// Block: HW_Const_Values

DATA_BLOCK HW_Const_Values
VERSION : 0.1
   NON_RETAIN
   VAR
      CU2_PN_IODevice : HW_DEVICE;
      CU2_PN : HW_INTERFACE;
      CU2_PN_Port_1 : HW_INTERFACE;
      CU2_PN_Port_2 : HW_INTERFACE;
      CU2_PN_585A1_ModuleAccessPoint : HW_SUBMODULE;
      CU2_PN_1190A1_ModuleAccessPoint : HW_SUBMODULE;
      CU2_PN_1300A1_ModuleAccessPoint : HW_SUBMODULE;
      CU2_PN_830A1_ModuleAccessPoint : HW_SUBMODULE;
      CU2_PN_1 : HW_INTERFACE;
      CU2_PN_Port_1_1 : HW_INTERFACE;
      CU2_PN_Port_2_1 : HW_INTERFACE;
      CU2_PN_2 : HW_INTERFACE;
      CU2_PN_Port_1_2 : HW_INTERFACE;
      CU2_PN_Port_2_2 : HW_INTERFACE;
      CU2_PN_3 : HW_INTERFACE;
      CU2_PN_Port_1_3 : HW_INTERFACE;
      CU2_PN_Port_2_3 : HW_INTERFACE;
      Local_PROFINET_interface_GBIT_3 : HW_INTERFACE;
      Local_PROFINET_interface_GBIT_3_Port_1 : HW_INTERFACE;
      Local_412A1 : HW_SUBMODULE;
      Local_413A1 : HW_SUBMODULE;
      Local_413A2 : HW_SUBMODULE;
      Local_414A1 : HW_SUBMODULE;
      Local_415A1 : HW_SUBMODULE;
      Local_415A2 : HW_SUBMODULE;
      HW_460A1_JB001_Proxy : HW_SUBMODULE;
      HW_460A1_JB001_IODevice : HW_DEVICE;
      HW_460A1_JB001_Head : HW_SUBMODULE;
      HW_460A1_JB001_460A1_X1 : HW_INTERFACE;
      HW_460A1_JB001_479A3 : HW_SUBMODULE;
      HW_460A1_JB001_479A4 : HW_SUBMODULE;
      HW_460A1_JB001_480A1 : HW_SUBMODULE;
      HW_460A1_JB001_480A2 : HW_SUBMODULE;
      HW_460A1_JB001_482A1 : HW_SUBMODULE;
      HW_460A1_JB001_482A2 : HW_SUBMODULE;
      HW_460A1_JB001_Server_module_1 : HW_SUBMODULE;
      HW_460A1_JB001_464A1 : HW_SUBMODULE;
      HW_460A1_JB001_470A2 : HW_SUBMODULE;
      HW_460A1_JB001_470A1 : HW_SUBMODULE;
      HW_460A1_JB001_463A1 : HW_SUBMODULE;
      HW_460A1_JB001_460A1_X1_Port_2 : HW_INTERFACE;
      HW_460A1_JB001_460A1_X1_Port_1 : HW_INTERFACE;
      HW_460A1_JB001_465A1 : HW_SUBMODULE;
      HW_460A1_JB001_468A1 : HW_SUBMODULE;
      HW_460A1_JB001_468A2 : HW_SUBMODULE;
      HW_460A1_JB001_468A3 : HW_SUBMODULE;
      HW_460A1_JB001_468A4 : HW_SUBMODULE;
      HW_460A1_JB001_468A5 : HW_SUBMODULE;
      HW_460A1_JB001_468A6 : HW_SUBMODULE;
      HW_460A1_JB001_468A7 : HW_SUBMODULE;
      HW_460A1_JB001_468A8 : HW_SUBMODULE;
      HW_460A1_JB001_471A1 : HW_SUBMODULE;
      HW_460A1_JB001_471A2 : HW_SUBMODULE;
      HW_460A1_JB001_472A1 : HW_SUBMODULE;
      HW_460A1_JB001_474A1 : HW_SUBMODULE;
      HW_460A1_JB001_474A2 : HW_SUBMODULE;
      HW_460A1_JB001_474A3 : HW_SUBMODULE;
      HW_460A1_JB001_474A4 : HW_SUBMODULE;
      HW_460A1_JB001_474A5 : HW_SUBMODULE;
      HW_460A1_JB001_474A6 : HW_SUBMODULE;
      HW_460A1_JB001_474A7 : HW_SUBMODULE;
      HW_460A1_JB001_474A8 : HW_SUBMODULE;
      HW_460A1_JB001_475A1 : HW_SUBMODULE;
      HW_460A1_JB001_475A2 : HW_SUBMODULE;
      HW_460A1_JB001_475A3 : HW_SUBMODULE;
      HW_460A1_JB001_475A4 : HW_SUBMODULE;
      HW_460A1_JB001_475A5 : HW_SUBMODULE;
      HW_460A1_JB001_475A6 : HW_SUBMODULE;
      HW_460A1_JB001_475A7 : HW_SUBMODULE;
      HW_460A1_JB001_475A8 : HW_SUBMODULE;
      HW_460A1_JB001_476A1 : HW_SUBMODULE;
      HW_460A1_JB001_476A2 : HW_SUBMODULE;
      HW_460A1_JB001_476A3 : HW_SUBMODULE;
      HW_460A1_JB001_476A4 : HW_SUBMODULE;
      HW_460A1_JB001_476A5 : HW_SUBMODULE;
      HW_460A1_JB001_476A6 : HW_SUBMODULE;
      HW_460A1_JB001_478A1 : HW_SUBMODULE;
      HW_460A1_JB001_478A2 : HW_SUBMODULE;
      HW_460A1_JB001_478A3 : HW_SUBMODULE;
      HW_460A1_JB001_478A4 : HW_SUBMODULE;
      HW_460A1_JB001_478A5 : HW_SUBMODULE;
      HW_460A1_JB001_478A6 : HW_SUBMODULE;
      HW_460A1_JB001_478A7 : HW_SUBMODULE;
      HW_460A1_JB001_478A8 : HW_SUBMODULE;
      HW_460A1_JB001_479A1 : HW_SUBMODULE;
      HW_460A1_JB001_479A2 : HW_SUBMODULE;
      HW_490A1_JB301_Proxy : HW_SUBMODULE;
      HW_490A1_JB301_IODevice : HW_DEVICE;
      HW_490A1_JB301_Head : HW_SUBMODULE;
      HW_490A1_JB301_PROFINET_interface : HW_INTERFACE;
      HW_490A1_JB301_495A2 : HW_SUBMODULE;
      HW_490A1_JB301_495A1 : HW_SUBMODULE;
      HW_490A1_JB301_PROFINET_interface_Port_2 : HW_INTERFACE;
      HW_490A1_JB301_PROFINET_interface_Port_1 : HW_INTERFACE;
      HW_510A1_JB302_Proxy : HW_SUBMODULE;
      HW_510A1_JB302_IODevice : HW_DEVICE;
      HW_510A1_JB302_Head : HW_SUBMODULE;
      HW_510A1_JB302_PROFINET_interface : HW_INTERFACE;
      HW_510A1_JB302_515A2 : HW_SUBMODULE;
      HW_510A1_JB302_515A1 : HW_SUBMODULE;
      HW_510A1_JB302_513A1 : HW_SUBMODULE;
      HW_510A1_JB302_512A1 : HW_SUBMODULE;
      HW_510A1_JB302_PROFINET_interface_Port_2 : HW_INTERFACE;
      HW_510A1_JB302_PROFINET_interface_Port_1 : HW_INTERFACE;
      HW_530A1_JB305_Proxy : HW_SUBMODULE;
      HW_530A1_JB305_IODevice : HW_DEVICE;
      HW_530A1_JB305_Head : HW_SUBMODULE;
      HW_530A1_JB305_PROFINET_interface : HW_INTERFACE;
      HW_530A1_JB305_542A3 : HW_SUBMODULE;
      HW_530A1_JB305_542A2 : HW_SUBMODULE;
      HW_530A1_JB305_542A1 : HW_SUBMODULE;
      HW_530A1_JB305_540A2 : HW_SUBMODULE;
      HW_530A1_JB305_540A1 : HW_SUBMODULE;
      HW_530A1_JB305_538A6 : HW_SUBMODULE;
      HW_530A1_JB305_538A5 : HW_SUBMODULE;
      HW_530A1_JB305_538A4 : HW_SUBMODULE;
      HW_530A1_JB305_538A3 : HW_SUBMODULE;
      HW_530A1_JB305_538A2 : HW_SUBMODULE;
      HW_530A1_JB305_538A1 : HW_SUBMODULE;
      HW_530A1_JB305_537A1 : HW_SUBMODULE;
      HW_530A1_JB305_536A1 : HW_SUBMODULE;
      HW_530A1_JB305_535A2 : HW_SUBMODULE;
      HW_530A1_JB305_535A1 : HW_SUBMODULE;
      HW_530A1_JB305_533A1 : HW_SUBMODULE;
      HW_530A1_JB305_PROFINET_interface_Port_2 : HW_INTERFACE;
      HW_530A1_JB305_PROFINET_interface_Port_1 : HW_INTERFACE;
      HW_550A1_JB306_Proxy : HW_SUBMODULE;
      HW_550A1_JB306_IODevice : HW_DEVICE;
      HW_550A1_JB306_Head : HW_SUBMODULE;
      HW_550A1_JB306_PROFINET_interface : HW_INTERFACE;
      HW_550A1_JB306_562A3 : HW_SUBMODULE;
      HW_550A1_JB306_562A2 : HW_SUBMODULE;
      HW_550A1_JB306_562A1 : HW_SUBMODULE;
      HW_550A1_JB306_560A2 : HW_SUBMODULE;
      HW_550A1_JB306_560A1 : HW_SUBMODULE;
      HW_550A1_JB306_558A6 : HW_SUBMODULE;
      HW_550A1_JB306_558A5 : HW_SUBMODULE;
      HW_550A1_JB306_558A4 : HW_SUBMODULE;
      HW_550A1_JB306_558A3 : HW_SUBMODULE;
      HW_550A1_JB306_558A2 : HW_SUBMODULE;
      HW_550A1_JB306_558A1 : HW_SUBMODULE;
      HW_550A1_JB306_556A1 : HW_SUBMODULE;
      HW_550A1_JB306_555A1 : HW_SUBMODULE;
      HW_550A1_JB306_552A1 : HW_SUBMODULE;
      HW_550A1_JB306_PROFINET_interface_Port_2 : HW_INTERFACE;
      HW_550A1_JB306_PROFINET_interface_Port_1 : HW_INTERFACE;
      CU1_PN_IODevice : HW_DEVICE;
      CU1_PN : HW_INTERFACE;
      CU1_PN_Port_1 : HW_INTERFACE;
      CU1_PN_Port_2 : HW_INTERFACE;
      CU1_PN_580A1_ModuleAccessPoint : HW_SUBMODULE;
      CU1_PN_740A1_1_ModuleAccessPoint : HW_SUBMODULE;
      CU1_PN_740A1_2_ModuleAccessPoint : HW_SUBMODULE;
      CU1_PN_690A1_1_ModuleAccessPoint : HW_SUBMODULE;
      CU1_PN_690A1_2_ModuleAccessPoint : HW_SUBMODULE;
      CU1_PN_890A1_1_ModuleAccessPoint : HW_SUBMODULE;
      CU1_PN_890A1_2_ModuleAccessPoint : HW_SUBMODULE;
      CU1_PN_1 : HW_INTERFACE;
      CU1_PN_Port_1_1 : HW_INTERFACE;
      CU1_PN_Port_2_1 : HW_INTERFACE;
      CU1_PN_2 : HW_INTERFACE;
      CU1_PN_Port_1_2 : HW_INTERFACE;
      CU1_PN_Port_2_2 : HW_INTERFACE;
      CU1_PN_3 : HW_INTERFACE;
      CU1_PN_Port_1_3 : HW_INTERFACE;
      CU1_PN_Port_2_3 : HW_INTERFACE;
      CU3_PROFINET_interface_IODevice : HW_DEVICE;
      CU3_PROFINET_interface : HW_INTERFACE;
      CU3_PROFINET_interface_Port_1 : HW_INTERFACE;
      CU3_PROFINET_interface_Port_2 : HW_INTERFACE;
      CU3_PROFINET_interface_590A1_ModuleAccessPoint : HW_SUBMODULE;
      CU3_PROFINET_interface_590A1_SIEMENS_telegram_393 : HW_SUBMODULE;
      CU3_PROFINET_interface_1410A1_1_ModuleAccessPoint : HW_SUBMODULE;
      CU3_PROFINET_interface_1410A1_1_PROFIsafe_telegram_30 : HW_SUBMODULE;
      CU3_PROFINET_interface_1410A1_2_ModuleAccessPoint : HW_SUBMODULE;
      CU3_PROFINET_interface_1410A1_2_PROFIsafe_telegram_30 : HW_SUBMODULE;
      CU3_PROFINET_interface_1430A1_1_ModuleAccessPoint : HW_SUBMODULE;
      CU3_PROFINET_interface_1430A1_1_PROFIsafe_telegram_30 : HW_SUBMODULE;
      CU3_PROFINET_interface_1430A1_2_ModuleAccessPoint : HW_SUBMODULE;
      CU3_PROFINET_interface_1430A1_2_PROFIsafe_telegram_30 : HW_SUBMODULE;
      CU3_PROFINET_interface_1260A1_1_ModuleAccessPoint : HW_SUBMODULE;
      CU3_PROFINET_interface_1260A1_1_PROFIsafe_telegram_30 : HW_SUBMODULE;
      CU3_PROFINET_interface_1260A1_2_ModuleAccessPoint : HW_SUBMODULE;
      CU3_PROFINET_interface_1260A1_2_PROFIsafe_telegram_30 : HW_SUBMODULE;
      CU3_PROFINET_interface_1 : HW_INTERFACE;
      CU3_PROFINET_interface_Port_1_1 : HW_INTERFACE;
      CU3_PROFINET_interface_Port_2_1 : HW_INTERFACE;
      CU3_PROFINET_interface_2 : HW_INTERFACE;
      CU3_PROFINET_interface_Port_1_2 : HW_INTERFACE;
      CU3_PROFINET_interface_Port_2_2 : HW_INTERFACE;
      CU3_PROFINET_interface_3 : HW_INTERFACE;
      CU3_PROFINET_interface_Port_1_3 : HW_INTERFACE;
      CU3_PROFINET_interface_Port_2_3 : HW_INTERFACE;
      CU4_PN_IODevice : HW_DEVICE;
      CU4_PN : HW_INTERFACE;
      CU4_PN_Port_1 : HW_INTERFACE;
      CU4_PN_Port_2 : HW_INTERFACE;
      CU4_PN_595A1_ModuleAccessPoint : HW_SUBMODULE;
      CU4_PN_595A1_SIEMENS_telegram_393 : HW_SUBMODULE;
      CU4_PN_980A1_1_ModuleAccessPoint : HW_SUBMODULE;
      CU4_PN_980A1_1_PROFIsafe_telegram_30 : HW_SUBMODULE;
      CU4_PN_980A1_2_ModuleAccessPoint : HW_SUBMODULE;
      CU4_PN_980A1_2_PROFIsafe_telegram_30 : HW_SUBMODULE;
      CU4_PN_1030A1_1_ModuleAccessPoint : HW_SUBMODULE;
      CU4_PN_1030A1_1_PROFIsafe_telegram_30 : HW_SUBMODULE;
      CU4_PN_1030A1_2_ModuleAccessPoint : HW_SUBMODULE;
      CU4_PN_1030A1_2_PROFIsafe_telegram_30 : HW_SUBMODULE;
      CU4_PN_1070A1_1_ModuleAccessPoint : HW_SUBMODULE;
      CU4_PN_1070A1_1_PROFIsafe_telegram_30 : HW_SUBMODULE;
      CU4_PN_1070A1_2_ModuleAccessPoint : HW_SUBMODULE;
      CU4_PN_1070A1_2_PROFIsafe_telegram_30 : HW_SUBMODULE;
      CU4_PN_1 : HW_INTERFACE;
      CU4_PN_Port_1_1 : HW_INTERFACE;
      CU4_PN_Port_2_1 : HW_INTERFACE;
      CU4_PN_2 : HW_INTERFACE;
      CU4_PN_Port_1_2 : HW_INTERFACE;
      CU4_PN_Port_2_2 : HW_INTERFACE;
      CU4_PN_3 : HW_INTERFACE;
      CU4_PN_Port_1_3 : HW_INTERFACE;
      CU4_PN_Port_2_3 : HW_INTERFACE;
      CU5_PN_IODevice : HW_DEVICE;
      CU5_PN : HW_INTERFACE;
      CU5_PN_Port_1 : HW_INTERFACE;
      CU5_PN_Port_2 : HW_INTERFACE;
      CU5_PN_600A1_ModuleAccessPoint : HW_SUBMODULE;
      CU5_PN_600A1_SIEMENS_telegram_393 : HW_SUBMODULE;
      CU5_PN_1950A1_ModuleAccessPoint : HW_SUBMODULE;
      CU5_PN_1950A1_SIEMENS_telegram_111 : HW_SUBMODULE;
      CU5_PN_1950A1_PROFIsafe_telegram_30 : HW_SUBMODULE;
      CU5_PN_1480A1_1_ModuleAccessPoint : HW_SUBMODULE;
      CU5_PN_1480A1_1_PROFIsafe_telegram_30 : HW_SUBMODULE;
      CU5_PN_1480A1_2_ModuleAccessPoint : HW_SUBMODULE;
      CU5_PN_1480A1_2_PROFIsafe_telegram_30 : HW_SUBMODULE;
      CU5_PN_1560A1_1_ModuleAccessPoint : HW_SUBMODULE;
      CU5_PN_1560A1_1_SIEMENS_telegram_111 : HW_SUBMODULE;
      CU5_PN_1560A1_1_PROFIsafe_telegram_30 : HW_SUBMODULE;
      CU5_PN_1560A1_2_ModuleAccessPoint : HW_SUBMODULE;
      CU5_PN_1560A1_2_SIEMENS_telegram_111 : HW_SUBMODULE;
      CU5_PN_1560A1_2_PROFIsafe_telegram_30 : HW_SUBMODULE;
      CU5_PN_1 : HW_INTERFACE;
      CU5_PN_Port_1_1 : HW_INTERFACE;
      CU5_PN_Port_2_1 : HW_INTERFACE;
      CU5_PN_2 : HW_INTERFACE;
      CU5_PN_Port_1_2 : HW_INTERFACE;
      CU5_PN_Port_2_2 : HW_INTERFACE;
      CU5_PN_3 : HW_INTERFACE;
      CU5_PN_Port_1_3 : HW_INTERFACE;
      CU5_PN_Port_2_3 : HW_INTERFACE;
      CU6_PN_IODevice : HW_DEVICE;
      CU6_PN : HW_INTERFACE;
      CU6_PN_Port_1 : HW_INTERFACE;
      CU6_PN_Port_2 : HW_INTERFACE;
      CU6_PN_605A1_ModuleAccessPoint : HW_SUBMODULE;
      CU6_PN_605A1_SIEMENS_telegram_393 : HW_SUBMODULE;
      CU6_PN_1990A1_1_ModuleAccessPoint : HW_SUBMODULE;
      CU6_PN_1990A1_1_PROFIsafe_telegram_30 : HW_SUBMODULE;
      CU6_PN_1990A1_2_ModuleAccessPoint : HW_SUBMODULE;
      CU6_PN_1990A1_2_PROFIsafe_telegram_30 : HW_SUBMODULE;
      CU6_PN_2100A1_1_ModuleAccessPoint : HW_SUBMODULE;
      CU6_PN_2100A1_1_SIEMENS_telegram_1 : HW_SUBMODULE;
      CU6_PN_2100A1_1_PROFIsafe_telegram_30 : HW_SUBMODULE;
      CU6_PN_2100A1_2_ModuleAccessPoint : HW_SUBMODULE;
      CU6_PN_2100A1_2_SIEMENS_telegram_1 : HW_SUBMODULE;
      CU6_PN_2100A1_2_PROFIsafe_telegram_30 : HW_SUBMODULE;
      CU6_PN_1840A1_1_ModuleAccessPoint : HW_SUBMODULE;
      CU6_PN_1840A1_1_PROFIsafe_telegram_30 : HW_SUBMODULE;
      CU6_PN_1840A1_2_ModuleAccessPoint : HW_SUBMODULE;
      CU6_PN_1840A1_2_PROFIsafe_telegram_30 : HW_SUBMODULE;
      CU6_PN_1 : HW_INTERFACE;
      CU6_PN_Port_1_1 : HW_INTERFACE;
      CU6_PN_Port_2_1 : HW_INTERFACE;
      CU6_PN_2 : HW_INTERFACE;
      CU6_PN_Port_1_2 : HW_INTERFACE;
      CU6_PN_Port_2_2 : HW_INTERFACE;
      CU6_PN_3 : HW_INTERFACE;
      CU6_PN_Port_1_3 : HW_INTERFACE;
      CU6_PN_Port_2_3 : HW_INTERFACE;
      CU7_PN_IODevice : HW_DEVICE;
      CU7_PN : HW_INTERFACE;
      CU7_PN_Port_1 : HW_INTERFACE;
      CU7_PN_Port_2 : HW_INTERFACE;
      CU7_PN_610A1_ModuleAccessPoint : HW_SUBMODULE;
      CU7_PN_610A1_SIEMENS_telegram_393 : HW_SUBMODULE;
      CU7_PN_2310A1_1_ModuleAccessPoint : HW_SUBMODULE;
      CU7_PN_2310A1_1_SIEMENS_telegram_111 : HW_SUBMODULE;
      CU7_PN_2310A1_1_PROFIsafe_telegram_30 : HW_SUBMODULE;
      CU7_PN_2310A1_2_ModuleAccessPoint : HW_SUBMODULE;
      CU7_PN_2310A1_2_SIEMENS_telegram_111 : HW_SUBMODULE;
      CU7_PN_2310A1_2_PROFIsafe_telegram_30 : HW_SUBMODULE;
      CU7_PN_2260A1_1_ModuleAccessPoint : HW_SUBMODULE;
      CU7_PN_2260A1_1_PROFIsafe_telegram_30 : HW_SUBMODULE;
      CU7_PN_2260A1_2_ModuleAccessPoint : HW_SUBMODULE;
      CU7_PN_2260A1_2_PROFIsafe_telegram_30 : HW_SUBMODULE;
      CU7_PN_2140A1_1_ModuleAccessPoint : HW_SUBMODULE;
      CU7_PN_2140A1_1_SIEMENS_telegram_111 : HW_SUBMODULE;
      CU7_PN_2140A1_1_PROFIsafe_telegram_30 : HW_SUBMODULE;
      CU7_PN_2140A1_2_ModuleAccessPoint : HW_SUBMODULE;
      CU7_PN_2140A1_2_SIEMENS_telegram_111 : HW_SUBMODULE;
      CU7_PN_2140A1_2_PROFIsafe_telegram_30 : HW_SUBMODULE;
      CU7_PN_1 : HW_INTERFACE;
      CU7_PN_Port_1_1 : HW_INTERFACE;
      CU7_PN_Port_2_1 : HW_INTERFACE;
      CU7_PN_2 : HW_INTERFACE;
      CU7_PN_Port_1_2 : HW_INTERFACE;
      CU7_PN_Port_2_2 : HW_INTERFACE;
      CU7_PN_3 : HW_INTERFACE;
      CU7_PN_Port_1_3 : HW_INTERFACE;
      CU7_PN_Port_2_3 : HW_INTERFACE;
      CU8_PN_IODevice : HW_DEVICE;
      CU8_PN : HW_INTERFACE;
      CU8_PN_Port_1 : HW_INTERFACE;
      CU8_PN_Port_2 : HW_INTERFACE;
      CU8_PN_615A1_ModuleAccessPoint : HW_SUBMODULE;
      CU8_PN_615A1_SIEMENS_telegram_393 : HW_SUBMODULE;
      CU8_PN_2390A1_1_ModuleAccessPoint : HW_SUBMODULE;
      CU8_PN_2390A1_1_PROFIsafe_telegram_30 : HW_SUBMODULE;
      CU8_PN_2390A1_2_ModuleAccessPoint : HW_SUBMODULE;
      CU8_PN_2390A1_2_PROFIsafe_telegram_30 : HW_SUBMODULE;
      CU8_PN_2430A1_1_ModuleAccessPoint : HW_SUBMODULE;
      CU8_PN_2430A1_1_PROFIsafe_telegram_30 : HW_SUBMODULE;
      CU8_PN_2430A1_2_ModuleAccessPoint : HW_SUBMODULE;
      CU8_PN_2430A1_2_PROFIsafe_telegram_30 : HW_SUBMODULE;
      CU8_PN_2350A1_1_ModuleAccessPoint : HW_SUBMODULE;
      CU8_PN_2350A1_1_PROFIsafe_telegram_30 : HW_SUBMODULE;
      CU8_PN_2350A1_2_ModuleAccessPoint : HW_SUBMODULE;
      CU8_PN_2350A1_2_PROFIsafe_telegram_30 : HW_SUBMODULE;
      CU8_PN_640A1_ModuleAccessPoint : HW_SUBMODULE;
      CU8_PN_640A1_SIEMENS_telegram_370 : HW_SUBMODULE;
      CU8_PN_1 : HW_INTERFACE;
      CU8_PN_Port_1_1 : HW_INTERFACE;
      CU8_PN_Port_2_1 : HW_INTERFACE;
      CU8_PN_2 : HW_INTERFACE;
      CU8_PN_Port_1_2 : HW_INTERFACE;
      CU8_PN_Port_2_2 : HW_INTERFACE;
      CU8_PN_3 : HW_INTERFACE;
      CU8_PN_Port_1_3 : HW_INTERFACE;
      CU8_PN_Port_2_3 : HW_INTERFACE;
      HW_1008P1_Proxy : HW_SUBMODULE;
      HW_1008P1_IODevice : HW_DEVICE;
      HW_1008P1_Interface : HW_INTERFACE;
      HW_1008P1_Interface_Port_1 : HW_INTERFACE;
      HW_1008P1_Interface_Port_2 : HW_INTERFACE;
      HW_1008P1_Head : HW_SUBMODULE;
      HW_1008P1_EO_Multiturn_1 : HW_SUBMODULE;
      HW_1008P1_Telegram_81_DI_DO : HW_SUBMODULE;
      HW_1008P1_EO_Multiturn_1_Parameter_Access_Point : HW_SUBMODULE;
      HW_1004P1_Proxy : HW_SUBMODULE;
      HW_1004P1_IODevice : HW_DEVICE;
      HW_1004P1_Interface : HW_INTERFACE;
      HW_1004P1_Interface_Port_1 : HW_INTERFACE;
      HW_1004P1_Interface_Port_2 : HW_INTERFACE;
      HW_1004P1_Head : HW_SUBMODULE;
      HW_1004P1_EO_Multiturn_1 : HW_SUBMODULE;
      HW_1004P1_Telegram_81_DI_DO : HW_SUBMODULE;
      HW_1004P1_EO_Multiturn_1_Parameter_Access_Point : HW_SUBMODULE;
      HW_994P1_Proxy : HW_SUBMODULE;
      HW_994P1_IODevice : HW_DEVICE;
      HW_994P1_Interface : HW_INTERFACE;
      HW_994P1_Interface_Port_1 : HW_INTERFACE;
      HW_994P1_Interface_Port_2 : HW_INTERFACE;
      HW_994P1_Head : HW_SUBMODULE;
      HW_994P1_EO_Multiturn_1 : HW_SUBMODULE;
      HW_994P1_Telegram_81_DI_DO : HW_SUBMODULE;
      HW_994P1_EO_Multiturn_1_Parameter_Access_Point : HW_SUBMODULE;
      HW_984P1_Proxy : HW_SUBMODULE;
      HW_984P1_IODevice : HW_DEVICE;
      HW_984P1_Interface : HW_INTERFACE;
      HW_984P1_Interface_Port_1 : HW_INTERFACE;
      HW_984P1_Interface_Port_2 : HW_INTERFACE;
      HW_984P1_Head : HW_SUBMODULE;
      HW_984P1_EO_Multiturn_1 : HW_SUBMODULE;
      HW_984P1_Telegram_81_DI_DO : HW_SUBMODULE;
      HW_984P1_EO_Multiturn_1_Parameter_Access_Point : HW_SUBMODULE;
      HW_1868P1_Proxy : HW_SUBMODULE;
      HW_1868P1_IODevice : HW_DEVICE;
      HW_1868P1_Interface : HW_INTERFACE;
      HW_1868P1_Interface_Port_1 : HW_INTERFACE;
      HW_1868P1_Interface_Port_2 : HW_INTERFACE;
      HW_1868P1_Head : HW_SUBMODULE;
      HW_1868P1_EO_Multiturn_1 : HW_SUBMODULE;
      HW_1868P1_Telegram_81_DI_DO : HW_SUBMODULE;
      HW_1868P1_EO_Multiturn_1_Parameter_Access_Point : HW_SUBMODULE;
      HW_1863P1_Proxy : HW_SUBMODULE;
      HW_1863P1_IODevice : HW_DEVICE;
      HW_1863P1_Interface : HW_INTERFACE;
      HW_1863P1_Interface_Port_1 : HW_INTERFACE;
      HW_1863P1_Interface_Port_2 : HW_INTERFACE;
      HW_1863P1_Head : HW_SUBMODULE;
      HW_1863P1_EO_Multiturn_1 : HW_SUBMODULE;
      HW_1863P1_Telegram_81_DI_DO : HW_SUBMODULE;
      HW_1863P1_EO_Multiturn_1_Parameter_Access_Point : HW_SUBMODULE;
      HW_1858P1_Proxy : HW_SUBMODULE;
      HW_1858P1_IODevice : HW_DEVICE;
      HW_1858P1_Interface : HW_INTERFACE;
      HW_1858P1_Interface_Port_1 : HW_INTERFACE;
      HW_1858P1_Interface_Port_2 : HW_INTERFACE;
      HW_1858P1_Head : HW_SUBMODULE;
      HW_1858P1_EO_Multiturn_1 : HW_SUBMODULE;
      HW_1858P1_Telegram_81_DI_DO : HW_SUBMODULE;
      HW_1858P1_EO_Multiturn_1_Parameter_Access_Point : HW_SUBMODULE;
      HW_1853P1_Proxy : HW_SUBMODULE;
      HW_1853P1_IODevice : HW_DEVICE;
      HW_1853P1_Interface : HW_INTERFACE;
      HW_1853P1_Interface_Port_1 : HW_INTERFACE;
      HW_1853P1_Interface_Port_2 : HW_INTERFACE;
      HW_1853P1_Head : HW_SUBMODULE;
      HW_1853P1_EO_Multiturn_1 : HW_SUBMODULE;
      HW_1853P1_Telegram_81_DI_DO : HW_SUBMODULE;
      HW_1853P1_EO_Multiturn_1_Parameter_Access_Point : HW_SUBMODULE;
      HW_1844P1_Proxy : HW_SUBMODULE;
      HW_1844P1_IODevice : HW_DEVICE;
      HW_1844P1_Interface : HW_INTERFACE;
      HW_1844P1_Interface_Port_1 : HW_INTERFACE;
      HW_1844P1_Interface_Port_2 : HW_INTERFACE;
      HW_1844P1_Head : HW_SUBMODULE;
      HW_1844P1_EO_Multiturn_1 : HW_SUBMODULE;
      HW_1844P1_Telegram_81_DI_DO : HW_SUBMODULE;
      HW_1844P1_EO_Multiturn_1_Parameter_Access_Point : HW_SUBMODULE;
      HW_1044P1_Proxy : HW_SUBMODULE;
      HW_1044P1_IODevice : HW_DEVICE;
      HW_1044P1_Interface : HW_INTERFACE;
      HW_1044P1_Interface_Port_1 : HW_INTERFACE;
      HW_1044P1_Interface_Port_2 : HW_INTERFACE;
      HW_1044P1_Head : HW_SUBMODULE;
      HW_1044P1_EO_Multiturn_1 : HW_SUBMODULE;
      HW_1044P1_Telegram_81_DI_DO : HW_SUBMODULE;
      HW_1044P1_EO_Multiturn_1_Parameter_Access_Point : HW_SUBMODULE;
      HW_1034P1_Proxy : HW_SUBMODULE;
      HW_1034P1_IODevice : HW_DEVICE;
      HW_1034P1_Interface : HW_INTERFACE;
      HW_1034P1_Interface_Port_1 : HW_INTERFACE;
      HW_1034P1_Interface_Port_2 : HW_INTERFACE;
      HW_1034P1_Head : HW_SUBMODULE;
      HW_1034P1_EO_Multiturn_1 : HW_SUBMODULE;
      HW_1034P1_Telegram_81_DI_DO : HW_SUBMODULE;
      HW_1034P1_EO_Multiturn_1_Parameter_Access_Point : HW_SUBMODULE;
      HW_1918P1_Proxy : HW_SUBMODULE;
      HW_1918P1_IODevice : HW_DEVICE;
      HW_1918P1_Interface : HW_INTERFACE;
      HW_1918P1_Interface_Port_1 : HW_INTERFACE;
      HW_1918P1_Interface_Port_2 : HW_INTERFACE;
      HW_1918P1_Head : HW_SUBMODULE;
      HW_1918P1_EO_Multiturn_1 : HW_SUBMODULE;
      HW_1918P1_Telegram_81_DI_DO : HW_SUBMODULE;
      HW_1918P1_EO_Multiturn_1_Parameter_Access_Point : HW_SUBMODULE;
      HW_1093P1_Proxy : HW_SUBMODULE;
      HW_1093P1_IODevice : HW_DEVICE;
      HW_1093P1_Interface : HW_INTERFACE;
      HW_1093P1_Interface_Port_1 : HW_INTERFACE;
      HW_1093P1_Interface_Port_2 : HW_INTERFACE;
      HW_1093P1_Head : HW_SUBMODULE;
      HW_1093P1_EO_Multiturn_1 : HW_SUBMODULE;
      HW_1093P1_Telegram_81_DI_DO : HW_SUBMODULE;
      HW_1093P1_EO_Multiturn_1_Parameter_Access_Point : HW_SUBMODULE;
      HW_1913P1_Proxy : HW_SUBMODULE;
      HW_1913P1_IODevice : HW_DEVICE;
      HW_1913P1_Interface : HW_INTERFACE;
      HW_1913P1_Interface_Port_1 : HW_INTERFACE;
      HW_1913P1_Interface_Port_2 : HW_INTERFACE;
      HW_1913P1_Head : HW_SUBMODULE;
      HW_1913P1_EO_Multiturn_1 : HW_SUBMODULE;
      HW_1913P1_Telegram_81_DI_DO : HW_SUBMODULE;
      HW_1913P1_EO_Multiturn_1_Parameter_Access_Point : HW_SUBMODULE;
      HW_1908P1_Proxy : HW_SUBMODULE;
      HW_1908P1_IODevice : HW_DEVICE;
      HW_1908P1_Interface : HW_INTERFACE;
      HW_1908P1_Interface_Port_1 : HW_INTERFACE;
      HW_1908P1_Interface_Port_2 : HW_INTERFACE;
      HW_1908P1_Head : HW_SUBMODULE;
      HW_1908P1_EO_Multiturn_1 : HW_SUBMODULE;
      HW_1908P1_Telegram_81_DI_DO : HW_SUBMODULE;
      HW_1908P1_EO_Multiturn_1_Parameter_Access_Point : HW_SUBMODULE;
      HW_1088P1_Proxy : HW_SUBMODULE;
      HW_1088P1_IODevice : HW_DEVICE;
      HW_1088P1_Interface : HW_INTERFACE;
      HW_1088P1_Interface_Port_1 : HW_INTERFACE;
      HW_1088P1_Interface_Port_2 : HW_INTERFACE;
      HW_1088P1_Head : HW_SUBMODULE;
      HW_1088P1_EO_Multiturn_1 : HW_SUBMODULE;
      HW_1088P1_Telegram_81_DI_DO : HW_SUBMODULE;
      HW_1088P1_EO_Multiturn_1_Parameter_Access_Point : HW_SUBMODULE;
      HW_1074P1_Proxy : HW_SUBMODULE;
      HW_1074P1_IODevice : HW_DEVICE;
      HW_1074P1_Interface : HW_INTERFACE;
      HW_1074P1_Interface_Port_1 : HW_INTERFACE;
      HW_1074P1_Interface_Port_2 : HW_INTERFACE;
      HW_1074P1_Head : HW_SUBMODULE;
      HW_1074P1_EO_Multiturn_1 : HW_SUBMODULE;
      HW_1074P1_Telegram_81_DI_DO : HW_SUBMODULE;
      HW_1074P1_EO_Multiturn_1_Parameter_Access_Point : HW_SUBMODULE;
      HW_1903P1_Proxy : HW_SUBMODULE;
      HW_1903P1_IODevice : HW_DEVICE;
      HW_1903P1_Interface : HW_INTERFACE;
      HW_1903P1_Interface_Port_1 : HW_INTERFACE;
      HW_1903P1_Interface_Port_2 : HW_INTERFACE;
      HW_1903P1_Head : HW_SUBMODULE;
      HW_1903P1_EO_Multiturn_1 : HW_SUBMODULE;
      HW_1903P1_Telegram_81_DI_DO : HW_SUBMODULE;
      HW_1903P1_EO_Multiturn_1_Parameter_Access_Point : HW_SUBMODULE;
      HW_1143P1_Proxy : HW_SUBMODULE;
      HW_1143P1_IODevice : HW_DEVICE;
      HW_1143P1_Interface : HW_INTERFACE;
      HW_1143P1_Interface_Port_1 : HW_INTERFACE;
      HW_1143P1_Interface_Port_2 : HW_INTERFACE;
      HW_1143P1_Head : HW_SUBMODULE;
      HW_1143P1_EO_Multiturn_1 : HW_SUBMODULE;
      HW_1143P1_Telegram_81_DI_DO : HW_SUBMODULE;
      HW_1143P1_EO_Multiturn_1_Parameter_Access_Point : HW_SUBMODULE;
      HW_1138P1_Proxy : HW_SUBMODULE;
      HW_1138P1_IODevice : HW_DEVICE;
      HW_1138P1_Interface : HW_INTERFACE;
      HW_1138P1_Interface_Port_1 : HW_INTERFACE;
      HW_1138P1_Interface_Port_2 : HW_INTERFACE;
      HW_1138P1_Head : HW_SUBMODULE;
      HW_1138P1_EO_Multiturn_1 : HW_SUBMODULE;
      HW_1138P1_Telegram_81_DI_DO : HW_SUBMODULE;
      HW_1138P1_EO_Multiturn_1_Parameter_Access_Point : HW_SUBMODULE;
      HW_2264P1_Proxy : HW_SUBMODULE;
      HW_2264P1_IODevice : HW_DEVICE;
      HW_2264P1_Interface : HW_INTERFACE;
      HW_2264P1_Interface_Port_1 : HW_INTERFACE;
      HW_2264P1_Interface_Port_2 : HW_INTERFACE;
      HW_2264P1_Head : HW_SUBMODULE;
      HW_2264P1_EO_Multiturn_1 : HW_SUBMODULE;
      HW_2264P1_Telegram_81_DI_DO : HW_SUBMODULE;
      HW_2264P1_EO_Multiturn_1_Parameter_Access_Point : HW_SUBMODULE;
      HW_1124P1_Proxy : HW_SUBMODULE;
      HW_1124P1_IODevice : HW_DEVICE;
      HW_1124P1_Interface : HW_INTERFACE;
      HW_1124P1_Interface_Port_1 : HW_INTERFACE;
      HW_1124P1_Interface_Port_2 : HW_INTERFACE;
      HW_1124P1_Head : HW_SUBMODULE;
      HW_1124P1_EO_Multiturn_1 : HW_SUBMODULE;
      HW_1124P1_Telegram_81_DI_DO : HW_SUBMODULE;
      HW_1124P1_EO_Multiturn_1_Parameter_Access_Point : HW_SUBMODULE;
      HW_2284P1_Proxy : HW_SUBMODULE;
      HW_2284P1_IODevice : HW_DEVICE;
      HW_2284P1_Interface : HW_INTERFACE;
      HW_2284P1_Interface_Port_1 : HW_INTERFACE;
      HW_2284P1_Interface_Port_2 : HW_INTERFACE;
      HW_2284P1_Head : HW_SUBMODULE;
      HW_2284P1_EO_Multiturn_1 : HW_SUBMODULE;
      HW_2284P1_Telegram_81_DI_DO : HW_SUBMODULE;
      HW_2284P1_EO_Multiturn_1_Parameter_Access_Point : HW_SUBMODULE;
      HW_694P1_Proxy : HW_SUBMODULE;
      HW_694P1_IODevice : HW_DEVICE;
      HW_694P1_Interface : HW_INTERFACE;
      HW_694P1_Interface_Port_1 : HW_INTERFACE;
      HW_694P1_Interface_Port_2 : HW_INTERFACE;
      HW_694P1_Head : HW_SUBMODULE;
      HW_694P1_EO_Multiturn_1 : HW_SUBMODULE;
      HW_694P1_Telegram_81_DI_DO : HW_SUBMODULE;
      HW_694P1_EO_Multiturn_1_Parameter_Access_Point : HW_SUBMODULE;
      HW_2354P1_Proxy : HW_SUBMODULE;
      HW_2354P1_IODevice : HW_DEVICE;
      HW_2354P1_Interface : HW_INTERFACE;
      HW_2354P1_Interface_Port_1 : HW_INTERFACE;
      HW_2354P1_Interface_Port_2 : HW_INTERFACE;
      HW_2354P1_Head : HW_SUBMODULE;
      HW_2354P1_EO_Multiturn_1 : HW_SUBMODULE;
      HW_2354P1_Telegram_81_DI_DO : HW_SUBMODULE;
      HW_2354P1_EO_Multiturn_1_Parameter_Access_Point : HW_SUBMODULE;
      HW_894P1_Proxy : HW_SUBMODULE;
      HW_894P1_IODevice : HW_DEVICE;
      HW_894P1_Interface : HW_INTERFACE;
      HW_894P1_Interface_Port_1 : HW_INTERFACE;
      HW_894P1_Interface_Port_2 : HW_INTERFACE;
      HW_894P1_Head : HW_SUBMODULE;
      HW_894P1_EO_Multiturn_1 : HW_SUBMODULE;
      HW_894P1_Telegram_81_DI_DO : HW_SUBMODULE;
      HW_894P1_EO_Multiturn_1_Parameter_Access_Point : HW_SUBMODULE;
      HW_2374P1_Proxy : HW_SUBMODULE;
      HW_2374P1_IODevice : HW_DEVICE;
      HW_2374P1_Interface : HW_INTERFACE;
      HW_2374P1_Interface_Port_1 : HW_INTERFACE;
      HW_2374P1_Interface_Port_2 : HW_INTERFACE;
      HW_2374P1_Head : HW_SUBMODULE;
      HW_2374P1_EO_Multiturn_1 : HW_SUBMODULE;
      HW_2374P1_Telegram_81_DI_DO : HW_SUBMODULE;
      HW_2374P1_EO_Multiturn_1_Parameter_Access_Point : HW_SUBMODULE;
      HW_100A1_Proxy : HW_SUBMODULE;
      HW_100A1_IODevice : HW_DEVICE;
      HW_100A1_PN_IO : HW_INTERFACE;
      HW_100A1_PN_IO_Port_1 : HW_INTERFACE;
      HW_100A1_PN_IO_Port_2 : HW_INTERFACE;
      HW_100A1_Head : HW_SUBMODULE;
      HW_2394P1_Proxy : HW_SUBMODULE;
      HW_2394P1_IODevice : HW_DEVICE;
      HW_2394P1_Interface : HW_INTERFACE;
      HW_2394P1_Interface_Port_1 : HW_INTERFACE;
      HW_2394P1_Interface_Port_2 : HW_INTERFACE;
      HW_2394P1_Head : HW_SUBMODULE;
      HW_2394P1_EO_Multiturn_1 : HW_SUBMODULE;
      HW_2394P1_Telegram_81_DI_DO : HW_SUBMODULE;
      HW_2394P1_EO_Multiturn_1_Parameter_Access_Point : HW_SUBMODULE;
      HW_2404P1_Proxy : HW_SUBMODULE;
      HW_2404P1_IODevice : HW_DEVICE;
      HW_2404P1_Interface : HW_INTERFACE;
      HW_2404P1_Interface_Port_1 : HW_INTERFACE;
      HW_2404P1_Interface_Port_2 : HW_INTERFACE;
      HW_2404P1_Head : HW_SUBMODULE;
      HW_2404P1_EO_Multiturn_1 : HW_SUBMODULE;
      HW_2404P1_Telegram_81_DI_DO : HW_SUBMODULE;
      HW_2404P1_EO_Multiturn_1_Parameter_Access_Point : HW_SUBMODULE;
      HW_2434P1_Proxy : HW_SUBMODULE;
      HW_2434P1_IODevice : HW_DEVICE;
      HW_2434P1_Interface : HW_INTERFACE;
      HW_2434P1_Interface_Port_1 : HW_INTERFACE;
      HW_2434P1_Interface_Port_2 : HW_INTERFACE;
      HW_2434P1_Head : HW_SUBMODULE;
      HW_2434P1_EO_Multiturn_1 : HW_SUBMODULE;
      HW_2434P1_Telegram_81_DI_DO : HW_SUBMODULE;
      HW_2434P1_EO_Multiturn_1_Parameter_Access_Point : HW_SUBMODULE;
      HW_2464P1_Proxy : HW_SUBMODULE;
      HW_2464P1_IODevice : HW_DEVICE;
      HW_2464P1_Interface : HW_INTERFACE;
      HW_2464P1_Interface_Port_1 : HW_INTERFACE;
      HW_2464P1_Interface_Port_2 : HW_INTERFACE;
      HW_2464P1_Head : HW_SUBMODULE;
      HW_2464P1_EO_Multiturn_1 : HW_SUBMODULE;
      HW_2464P1_Telegram_81_DI_DO : HW_SUBMODULE;
      HW_2464P1_EO_Multiturn_1_Parameter_Access_Point : HW_SUBMODULE;
      HW_2104P1_Telegram_81_DI_DO : HW_SUBMODULE;
      HW_2184P1_Telegram_81_DI_DO : HW_SUBMODULE;
      HW_100A1_Voltage_L1_N_1 : HW_SUBMODULE;
      HW_100A1_Voltage_L2_N_1 : HW_SUBMODULE;
      HW_100A1_Voltage_L3_N_1 : HW_SUBMODULE;
      HW_100A1_Current_L1_1 : HW_SUBMODULE;
      HW_100A1_Current_L2_1 : HW_SUBMODULE;
      HW_100A1_Current_L3_1 : HW_SUBMODULE;
      HW_100A1_3_Ph_Average_Volt_L_L_1 : HW_SUBMODULE;
      HW_100A1_3_Ph_Average_Curr_1 : HW_SUBMODULE;
      HW_100A1_Total_Active_Power_1 : HW_SUBMODULE;
      HW_100A1_Total_Reac_Power_1 : HW_SUBMODULE;
      HW_100A1_Act_Energy_Imp_Tar_1_D_1 : HW_SUBMODULE;
      HW_100A1_Reac_En_Imp_Tar_1_D_1 : HW_SUBMODULE;
      HW_490A1_JB301_498A1 : HW_SUBMODULE;
      HW_490A1_JB301_498A2 : HW_SUBMODULE;
      HW_490A1_JB301_498A3 : HW_SUBMODULE;
      HW_490A1_JB301_500A1 : HW_SUBMODULE;
      HW_490A1_JB301_502A1 : HW_SUBMODULE;
      HW_490A1_JB301_502A2 : HW_SUBMODULE;
      HW_490A1_JB301_495A3 : HW_SUBMODULE;
      CU1_PN_580A1_SIEMENS_telegram_393 : HW_SUBMODULE;
      CU1_PN_580A1_SIEMENS_telegram_393_1 : HW_SUBMODULE;
      CU1_PN_740A1_1_PROFIsafe_telegram_30 : HW_SUBMODULE;
      CU1_PN_740A1_1_PROFIsafe_telegram_30_1 : HW_SUBMODULE;
      CU1_PN_740A1_2_PROFIsafe_telegram_30 : HW_SUBMODULE;
      CU1_PN_740A1_2_PROFIsafe_telegram_30_1 : HW_SUBMODULE;
      CU1_PN_690A1_1_PROFIsafe_telegram_30 : HW_SUBMODULE;
      CU1_PN_690A1_1_PROFIsafe_telegram_30_1 : HW_SUBMODULE;
      CU1_PN_690A1_2_PROFIsafe_telegram_30 : HW_SUBMODULE;
      CU1_PN_690A1_2_PROFIsafe_telegram_30_1 : HW_SUBMODULE;
      CU1_PN_890A1_1_PROFIsafe_telegram_30 : HW_SUBMODULE;
      CU1_PN_890A1_1_PROFIsafe_telegram_30_1 : HW_SUBMODULE;
      CU1_PN_890A1_2_PROFIsafe_telegram_30 : HW_SUBMODULE;
      CU1_PN_890A1_2_PROFIsafe_telegram_30_1 : HW_SUBMODULE;
      HW_490A1_JB301_Server_module_1 : HW_SUBMODULE;
      HW_510A1_JB302_518A1 : HW_SUBMODULE;
      HW_510A1_JB302_518A2 : HW_SUBMODULE;
      HW_510A1_JB302_518A3 : HW_SUBMODULE;
      HW_510A1_JB302_518A4 : HW_SUBMODULE;
      HW_510A1_JB302_518A5 : HW_SUBMODULE;
      HW_510A1_JB302_518A6 : HW_SUBMODULE;
      HW_510A1_JB302_518A7 : HW_SUBMODULE;
      HW_510A1_JB302_518A8 : HW_SUBMODULE;
      HW_510A1_JB302_519A1 : HW_SUBMODULE;
      HW_510A1_JB302_519A2 : HW_SUBMODULE;
      HW_510A1_JB302_519A3 : HW_SUBMODULE;
      HW_510A1_JB302_519A4 : HW_SUBMODULE;
      HW_510A1_JB302_519A5 : HW_SUBMODULE;
      HW_510A1_JB302_520A1 : HW_SUBMODULE;
      HW_510A1_JB302_520A2 : HW_SUBMODULE;
      HW_510A1_JB302_522A1 : HW_SUBMODULE;
      HW_510A1_JB302_522A2 : HW_SUBMODULE;
      HW_510A1_JB302_522A3 : HW_SUBMODULE;
      HW_510A1_JB302_522A4 : HW_SUBMODULE;
      HW_510A1_JB302_522A5 : HW_SUBMODULE;
      HW_510A1_JB302_522A6 : HW_SUBMODULE;
      HW_510A1_JB302_522A7 : HW_SUBMODULE;
      HW_510A1_JB302_522A8 : HW_SUBMODULE;
      HW_510A1_JB302_Server_module_1 : HW_SUBMODULE;
      HW_530A1_JB305_Server_module_1 : HW_SUBMODULE;
      HW_530A1_JB305_532A1 : HW_SUBMODULE;
      HW_550A1_JB306_Server_module_1 : HW_SUBMODULE;
      HU_Cytropac_Proxy : HW_SUBMODULE;
      HU_Cytropac_IODevice : HW_DEVICE;
      HU_Cytropac_PN_IO : HW_INTERFACE;
      HU_Cytropac_PN_IO_Port_1_RJ45 : HW_INTERFACE;
      HU_Cytropac_PN_IO_Port_2_RJ45 : HW_INTERFACE;
      HU_Cytropac_Head : HW_SUBMODULE;
      HU_Cytropac_Output_04_Words_1 : HW_SUBMODULE;
      HU_Cytropac_Input_08_Words_1 : HW_SUBMODULE;
      CU1_PN_740A1_1_Standard_telegram_1 : HW_SUBMODULE;
      CU1_PN_740A1_1_Standard_telegram_1_1 : HW_SUBMODULE;
      CU1_PN_740A1_2_Standard_telegram_1 : HW_SUBMODULE;
      CU1_PN_740A1_2_Standard_telegram_1_1 : HW_SUBMODULE;
      CU1_PN_690A1_1_Standard_telegram_1 : HW_SUBMODULE;
      CU1_PN_690A1_1_Standard_telegram_1_1 : HW_SUBMODULE;
      CU1_PN_690A1_2_Standard_telegram_1 : HW_SUBMODULE;
      CU1_PN_690A1_2_Standard_telegram_1_1 : HW_SUBMODULE;
      CU1_PN_890A1_1_Standard_telegram_1 : HW_SUBMODULE;
      CU1_PN_890A1_1_Standard_telegram_1_1 : HW_SUBMODULE;
      CU1_PN_890A1_2_Standard_telegram_1 : HW_SUBMODULE;
      CU1_PN_890A1_2_Standard_telegram_1_1 : HW_SUBMODULE;
      CU3_PROFINET_interface_1410A1_1_Standard_telegram_1 : HW_SUBMODULE;
      CU3_PROFINET_interface_1410A1_1_Standard_telegram_1_1 : HW_SUBMODULE;
      CU3_PROFINET_interface_1410A1_2_Standard_telegram_1 : HW_SUBMODULE;
      CU3_PROFINET_interface_1410A1_2_Standard_telegram_1_1 : HW_SUBMODULE;
      CU3_PROFINET_interface_1430A1_1_Standard_telegram_1 : HW_SUBMODULE;
      CU3_PROFINET_interface_1430A1_1_Standard_telegram_1_1 : HW_SUBMODULE;
      CU3_PROFINET_interface_1430A1_2_Standard_telegram_1 : HW_SUBMODULE;
      CU3_PROFINET_interface_1430A1_2_Standard_telegram_1_1 : HW_SUBMODULE;
      CU3_PROFINET_interface_1260A1_1_Standard_telegram_1 : HW_SUBMODULE;
      CU3_PROFINET_interface_1260A1_1_Standard_telegram_1_1 : HW_SUBMODULE;
      CU3_PROFINET_interface_1260A1_2_Standard_telegram_1 : HW_SUBMODULE;
      CU3_PROFINET_interface_1260A1_2_Standard_telegram_1_1 : HW_SUBMODULE;
      CU4_PN_980A1_1_Standard_telegram_1 : HW_SUBMODULE;
      CU4_PN_980A1_1_Standard_telegram_1_1 : HW_SUBMODULE;
      CU4_PN_980A1_2_Standard_telegram_1 : HW_SUBMODULE;
      CU4_PN_980A1_2_Standard_telegram_1_1 : HW_SUBMODULE;
      CU4_PN_1030A1_1_Standard_telegram_1 : HW_SUBMODULE;
      CU4_PN_1030A1_1_Standard_telegram_1_1 : HW_SUBMODULE;
      CU4_PN_1030A1_2_Standard_telegram_1 : HW_SUBMODULE;
      CU4_PN_1030A1_2_Standard_telegram_1_1 : HW_SUBMODULE;
      CU4_PN_1070A1_1_Standard_telegram_1 : HW_SUBMODULE;
      CU4_PN_1070A1_1_Standard_telegram_1_1 : HW_SUBMODULE;
      CU4_PN_1070A1_2_Standard_telegram_1 : HW_SUBMODULE;
      CU4_PN_1070A1_2_Standard_telegram_1_1 : HW_SUBMODULE;
      CU5_PN_1480A1_1_Standard_telegram_1 : HW_SUBMODULE;
      CU5_PN_1480A1_1_Standard_telegram_1_1 : HW_SUBMODULE;
      CU5_PN_1480A1_2_Standard_telegram_1 : HW_SUBMODULE;
      CU5_PN_1480A1_2_Standard_telegram_1_1 : HW_SUBMODULE;
      CU5_PN_1560A1_2_Standard_telegram_1_2 : HW_SUBMODULE;
      CU6_PN_1990A1_1_Standard_telegram_1 : HW_SUBMODULE;
      CU6_PN_1990A1_1_Standard_telegram_1_1 : HW_SUBMODULE;
      CU6_PN_1990A1_2_Standard_telegram_1 : HW_SUBMODULE;
      CU6_PN_1990A1_2_Standard_telegram_1_1 : HW_SUBMODULE;
      CU6_PN_1840A1_1_Standard_telegram_1 : HW_SUBMODULE;
      CU6_PN_1840A1_1_Standard_telegram_1_1 : HW_SUBMODULE;
      CU6_PN_1840A1_2_Standard_telegram_1 : HW_SUBMODULE;
      CU6_PN_1840A1_2_Standard_telegram_1_1 : HW_SUBMODULE;
      CU7_PN_2260A1_1_Standard_telegram_1 : HW_SUBMODULE;
      CU7_PN_2260A1_1_Standard_telegram_1_1 : HW_SUBMODULE;
      CU7_PN_2260A1_2_Standard_telegram_1 : HW_SUBMODULE;
      CU7_PN_2260A1_2_Standard_telegram_1_1 : HW_SUBMODULE;
      CU8_PN_2390A1_1_Standard_telegram_1 : HW_SUBMODULE;
      CU8_PN_2390A1_1_Standard_telegram_1_1 : HW_SUBMODULE;
      CU8_PN_2390A1_2_Standard_telegram_1 : HW_SUBMODULE;
      CU8_PN_2390A1_2_Standard_telegram_1_1 : HW_SUBMODULE;
      CU8_PN_2430A1_1_Standard_telegram_1 : HW_SUBMODULE;
      CU8_PN_2430A1_1_Standard_telegram_1_1 : HW_SUBMODULE;
      CU8_PN_2430A1_2_Standard_telegram_1 : HW_SUBMODULE;
      CU8_PN_2430A1_2_Standard_telegram_1_1 : HW_SUBMODULE;
      CU8_PN_2350A1_1_Standard_telegram_1 : HW_SUBMODULE;
      CU8_PN_2350A1_1_Standard_telegram_1_1 : HW_SUBMODULE;
      CU8_PN_2350A1_2_Standard_telegram_1 : HW_SUBMODULE;
      CU8_PN_2350A1_2_Standard_telegram_1_1 : HW_SUBMODULE;
      CU2_PN_585A1_SIEMENS_telegram_393 : HW_SUBMODULE;
      CU2_PN_585A1_SIEMENS_telegram_393_1 : HW_SUBMODULE;
      CU2_PN_1190A1_SIEMENS_telegram_106 : HW_SUBMODULE;
      CU2_PN_1190A1_SIEMENS_telegram_106_1 : HW_SUBMODULE;
      CU2_PN_1190A1_PROFIsafe_telegram_30 : HW_SUBMODULE;
      CU2_PN_1190A1_PROFIsafe_telegram_30_1 : HW_SUBMODULE;
      CU2_PN_1300A1_SIEMENS_telegram_106 : HW_SUBMODULE;
      CU2_PN_1300A1_SIEMENS_telegram_106_1 : HW_SUBMODULE;
      CU2_PN_1300A1_PROFIsafe_telegram_30 : HW_SUBMODULE;
      CU2_PN_1300A1_PROFIsafe_telegram_30_1 : HW_SUBMODULE;
      CU2_PN_830A1_SIEMENS_telegram_106 : HW_SUBMODULE;
      CU2_PN_830A1_SIEMENS_telegram_106_1 : HW_SUBMODULE;
      CU2_PN_830A1_PROFIsafe_telegram_30 : HW_SUBMODULE;
      CU2_PN_830A1_PROFIsafe_telegram_30_1 : HW_SUBMODULE;
      CU6_PN_2100A1_1_Standard_telegram_1 : HW_SUBMODULE;
      CU6_PN_2100A1_2_Standard_telegram_1 : HW_SUBMODULE;
      "dl-pn1_DL_PN1_1" : HW_SUBMODULE;
      "dl-pn1_IL-1000_Master" : HW_SUBMODULE;
      "dl-pn1_IL-1000_Slave" : HW_SUBMODULE;
   END_VAR

BEGIN
   // No initialization required
END_DATA_BLOCK
